(* PLC project  *)

PROGRAM LadderXml
  VAR
    Start : BOOL;
    Stop : BOOL;
    Override : BOOL;
    Motor : BOOL;
    Latched : BOOL;
  END_VAR

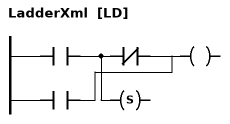
(* LD diagram, written out as Structured Text *)
 := ;
IF  THEN  := TRUE; END_IF;
END_PROGRAM
